INTERFACE I_ChunkedResponseData EXTENDS I_SessionData

PROPERTY PUBLIC SendComplete : BOOL
GET
END_GET
END_PROPERTY

METHOD PUBLIC SendNextChunk
VAR_INPUT
	Response : I_ServerResponse;
	Size : UDINT;
END_VAR
END_METHOD

PROPERTY SizeRemaining : UDINT
GET
END_GET
END_PROPERTY

END_INTERFACE

(* stored: Version 1.1.0.1, ProductVersion 3.1.4024.12
   Itf I_ChunkedResponseData: Id {94633d7f-cf45-4ad3-8a69-c634c872be06}
   Property SendComplete: Id {0feb97eb-9a15-4bda-bd86-f99d696bde80}
   Get Get: Id {185b6426-93a7-4307-8ab1-abae14604a3e}
   Method SendNextChunk: Id {34a950fd-f713-4e4b-9f81-4527c52406ca}
   Property SizeRemaining: Id {89b073cd-6d7c-4c68-98ba-56ea826e4a0e}
   Get Get: Id {1f0bca41-823c-4e54-b46b-db20e9d4b339} *)
